FUNCTION_BLOCK FB_ComponentTests
VAR_INPUT
END_VAR
VAR_OUTPUT
	fbTestsuite:			FB_Testsuite;
END_VAR
VAR
	fbComponent:				Tc3_Component.FB_Component;
END_VAR

fbTestsuite.P_Property.M_Add('object', 'FB_Component');
fbTestsuite.P_Property.M_Add('name', 'Peter Zerlauth');

fbTestsuite();

fbComponent();

CASE fbTestsuite.P_Testcase OF
	
	E_Testcase.Start:
		IF fbComponent.P_State = E_State.Aborted THEN
			fbComponent.M_Request(E_Request.Reset);
		ELSIF	fbComponent.P_State <> E_State.Idle THEN
			fbComponent.M_Request(E_Request.Abort);			
		END_IF

		fbTestsuite.P_Assert.M_Equals_STRING(TO_STRING(E_State.Idle), TO_STRING(fbComponent.P_State), 'P_State');
		fbTestsuite.M_Testcase('FB_Component', T#2S, 'fbComponent.M_Request(E_Request.Reset)', '', 10);	
		
	10:
		fbTestsuite.P_Assert.M_Equals_BOOL(TRUE, fbComponent.M_Request(E_Request.Start), 'M_Request(E_Request.Start)');	
		fbTestsuite.P_Assert.M_Equals_STRING(TO_STRING(E_State.Execute), TO_STRING(fbComponent.P_State), 'P_State');
		fbTestsuite.M_Testcase('FB_Component', T#2S, 'fbComponent.M_Request(E_Request.Reset)', '', 20);
		
	20:
		fbTestsuite.P_Assert.M_Equals_BOOL(TRUE, fbComponent.M_Request(E_Request.Abort), 'M_Request(E_Request.Abort)');	
		fbTestsuite.P_Assert.M_Equals_STRING(TO_STRING(E_State.Aborted), TO_STRING(fbComponent.P_State), 'P_State');
		fbTestsuite.M_Testcase('FB_Component', T#2S, 'fbComponent.M_Request(E_Request.Abort)', '', 30);

	30:
		fbTestsuite.P_Assert.M_Equals_BOOL(TRUE, fbComponent.M_Request(E_Request.Reset), 'M_Request(E_Request.Reset)');	
		fbTestsuite.P_Assert.M_Equals_STRING(TO_STRING(E_State.Idle), TO_STRING(fbComponent.P_State), 'P_State');
		fbTestsuite.M_Testcase('FB_Component', T#2S, 'fbComponent.M_Request(E_Request.Reset)', '', 40);

	40:
		fbTestsuite.P_Assert.M_Equals_BOOL(TRUE, fbComponent.M_Request(E_Request.Start), 'M_Request(E_Request.Start)');	
		fbTestsuite.P_Assert.M_Equals_STRING(TO_STRING(E_State.Execute), TO_STRING(fbComponent.P_State), 'P_State');
		fbTestsuite.M_Testcase('FB_Component', T#2S, 'fbComponent.M_Request(E_Request.Reset)', '', 50);
		
	50:
		fbTestsuite.P_Assert.M_Equals_BOOL(TRUE, fbComponent.M_Request(E_Request.Stop), 'M_Request(E_Request.Stop)');	
		fbTestsuite.P_Assert.M_Equals_STRING(TO_STRING(E_State.Stopped), TO_STRING(fbComponent.P_State), 'P_State');
		fbTestsuite.M_Testcase('FB_Component', T#2S, 'fbComponent.M_Request(E_Request.Stop)', '', 60);
		
	60:
		fbTestsuite.P_Assert.M_Equals_BOOL(TRUE, fbComponent.M_Request(E_Request.Reset), 'M_Request(E_Request.Reset)');	
		fbTestsuite.P_Assert.M_Equals_STRING(TO_STRING(E_State.Idle), TO_STRING(fbComponent.P_State), 'P_State');
		fbTestsuite.M_Testcase('FB_Component', T#2S, 'fbComponent.M_Request(E_Request.Reset)', '', 70);
		
	70:
		fbComponent.P_Event.M_Abort('Abort', 1);
		fbTestsuite.P_Assert.M_Equals_STRING(TO_STRING(E_State.Aborted), TO_STRING(fbComponent.P_State), 'P_State');
		fbTestsuite.M_Testcase('FB_Component', T#2S, 'fbComponent.P_Event.M_Abort(Abort, 1)', '', E_Testcase.Done);		
		
		
	E_Testcase.Done:
		;
END_CASE

END_FUNCTION_BLOCK

(* stored: Version 1.1.0.1
   POU FB_ComponentTests: Id {9c2d8e9a-6b38-0ce4-1e25-f4086cd07082}, SpecialFunc None *)
